(* IEC 61131-3 sources: 2026_Projet_YGO_ExcavatriceDragage/TOOLS/TEST_AUTO_CI/WORKING_COPY/tests (part 2) *)

(* ---- test_fb_cycle_negative.st ---- *)
SETUP
VAR
    FB : FB_Cycle;
    SampleCount : INT := 0;
END_VAR
END_SETUP

(* =====================================================================
   Harnais de TESTS NÉGATIFS — exécuté sur CODE/G_CYCLE/FB_Cycle.st (ORIGINAL).
   Chaque test DOIT ÉCHOUER sur l'original pour prouver la présence du défaut.
   Exclus de la suite verte (tests négatifs, exigence T3/T4 plan T171).
   ===================================================================== *)

TEST 'NEG-F1 : X11 ouverture benne commandee (doit ECHOUER sur original)'
    (* Atteindre X11 puis vérifier que BucketCmd.Open est TRUE quand le manche est défléchi.
       Sur l'original (read-before-write), Open reste FALSE -> ce test échoue. *)
    (* X0 -> X1 *)
    FB(Enable := TRUE, Reset := FALSE, PowerContactorEngaged := TRUE, Mode := E_Mode.SEMI_AUTO,
       DeadmanArmed := TRUE, CycleMotionPermit := TRUE, HeartbeatIhmOk := TRUE,
       StartCycle := TRUE, SelTarget := 3, SetDepthM := -10.0, SetOffsetM := 0.0,
       LimitLegalDepthM := -10.5, CableLimitM1AscentM := 7.0,
       SpeedMismatchThresholdMps := 0.0, SpeedMismatchTimeout := T#0ms,
       HomedM1 := TRUE, HomedM2 := TRUE, TopPositionSensor := TRUE, HomingRequest := FALSE,
       M1_CablePosM := 7.0, M2_CablePosM := 7.0, M1_MeasuredSpeedMps := 0.0, M2_MeasuredSpeedMps := 0.0,
       KoboldContactFond := FALSE, WinchSyncError := FALSE, WinchSyncDeltaM := 0.0,
       Translation_At_P1 := FALSE, Translation_At_Tremie := FALSE, Translation_At_Maintenance := FALSE,
       Translation_Busy := FALSE, Translation_Done := FALSE,
       Benne_Busy := FALSE, Benne_Done := FALSE, Benne_IsOpen := FALSE, Benne_IsClosed := TRUE, Benne_IsRoughlyClosed := TRUE,
       SampleCount := SampleCount);
    (* X1 -> X2 *)
    FB(Enable := TRUE, Reset := FALSE, PowerContactorEngaged := TRUE, Mode := E_Mode.SEMI_AUTO,
       DeadmanArmed := TRUE, CycleMotionPermit := TRUE, HeartbeatIhmOk := TRUE,
       StartCycle := FALSE, SelTarget := 3, SetDepthM := -10.0, SetOffsetM := 0.0,
       LimitLegalDepthM := -10.5, CableLimitM1AscentM := 7.0,
       SpeedMismatchThresholdMps := 0.0, SpeedMismatchTimeout := T#0ms,
       HomedM1 := TRUE, HomedM2 := TRUE, TopPositionSensor := TRUE, HomingRequest := FALSE,
       M1_CablePosM := 7.0, M2_CablePosM := 7.0, M1_MeasuredSpeedMps := 0.0, M2_MeasuredSpeedMps := 0.0,
       KoboldContactFond := FALSE, WinchSyncError := FALSE, WinchSyncDeltaM := 0.0,
       Translation_At_P1 := FALSE, Translation_At_Tremie := FALSE, Translation_At_Maintenance := FALSE,
       Translation_Busy := FALSE, Translation_Done := FALSE,
       Benne_Busy := FALSE, Benne_Done := FALSE, Benne_IsOpen := FALSE, Benne_IsClosed := TRUE, Benne_IsRoughlyClosed := TRUE,
       SampleCount := SampleCount);
    (* X2 -> X3 *)
    FB(Enable := TRUE, Reset := FALSE, PowerContactorEngaged := TRUE, Mode := E_Mode.SEMI_AUTO,
       DeadmanArmed := TRUE, CycleMotionPermit := TRUE, HeartbeatIhmOk := TRUE,
       StartCycle := FALSE, SelTarget := 3, SetDepthM := -10.0, SetOffsetM := 0.0,
       LimitLegalDepthM := -10.5, CableLimitM1AscentM := 7.0,
       SpeedMismatchThresholdMps := 0.0, SpeedMismatchTimeout := T#0ms,
       HomedM1 := TRUE, HomedM2 := TRUE, TopPositionSensor := TRUE, HomingRequest := FALSE,
       M1_CablePosM := 7.0, M2_CablePosM := 7.0, M1_MeasuredSpeedMps := 0.0, M2_MeasuredSpeedMps := 0.0,
       KoboldContactFond := FALSE, WinchSyncError := FALSE, WinchSyncDeltaM := 0.0,
       Translation_At_P1 := TRUE, Translation_At_Tremie := FALSE, Translation_At_Maintenance := FALSE,
       Translation_Busy := FALSE, Translation_Done := TRUE,
       Benne_Busy := FALSE, Benne_Done := FALSE, Benne_IsOpen := FALSE, Benne_IsClosed := TRUE, Benne_IsRoughlyClosed := TRUE,
       SampleCount := SampleCount);
    (* X3 -> X4 *)
    FB(Enable := TRUE, Reset := FALSE, PowerContactorEngaged := TRUE, Mode := E_Mode.SEMI_AUTO,
       DeadmanArmed := TRUE, CycleMotionPermit := TRUE, HeartbeatIhmOk := TRUE,
       StartCycle := FALSE, SelTarget := 3, SetDepthM := -10.0, SetOffsetM := 0.0,
       LimitLegalDepthM := -10.5, CableLimitM1AscentM := 7.0,
       SpeedMismatchThresholdMps := 0.0, SpeedMismatchTimeout := T#0ms,
       HomedM1 := TRUE, HomedM2 := TRUE, TopPositionSensor := TRUE, HomingRequest := FALSE,
       M1_CablePosM := 7.0, M2_CablePosM := 7.0, M1_MeasuredSpeedMps := 0.0, M2_MeasuredSpeedMps := 0.0,
       KoboldContactFond := FALSE, WinchSyncError := FALSE, WinchSyncDeltaM := 0.0,
       Translation_At_P1 := TRUE, Translation_At_Tremie := FALSE, Translation_At_Maintenance := FALSE,
       Translation_Busy := FALSE, Translation_Done := TRUE,
       Benne_Busy := FALSE, Benne_Done := FALSE, Benne_IsOpen := TRUE, Benne_IsClosed := FALSE, Benne_IsRoughlyClosed := FALSE,
       SampleCount := SampleCount);
    (* X4 -> X5 *)
    FB(Enable := TRUE, Reset := FALSE, PowerContactorEngaged := TRUE, Mode := E_Mode.SEMI_AUTO,
       DeadmanArmed := TRUE, CycleMotionPermit := TRUE, HeartbeatIhmOk := TRUE,
       StartCycle := FALSE, SelTarget := 3, SetDepthM := -10.0, SetOffsetM := 0.0,
       LimitLegalDepthM := -10.5, CableLimitM1AscentM := 7.0,
       SpeedMismatchThresholdMps := 0.0, SpeedMismatchTimeout := T#0ms,
       HomedM1 := TRUE, HomedM2 := TRUE, TopPositionSensor := TRUE, HomingRequest := FALSE,
       M1_CablePosM := -10.0, M2_CablePosM := -10.0, M1_MeasuredSpeedMps := 0.0, M2_MeasuredSpeedMps := 0.0,
       KoboldContactFond := TRUE, WinchSyncError := FALSE, WinchSyncDeltaM := 0.0,
       Translation_At_P1 := TRUE, Translation_At_Tremie := FALSE, Translation_At_Maintenance := FALSE,
       Translation_Busy := FALSE, Translation_Done := TRUE,
       Benne_Busy := FALSE, Benne_Done := FALSE, Benne_IsOpen := TRUE, Benne_IsClosed := FALSE, Benne_IsRoughlyClosed := FALSE,
       SampleCount := SampleCount);
    (* X5 -> X6 *)
    FB(Enable := TRUE, Reset := FALSE, PowerContactorEngaged := TRUE, Mode := E_Mode.SEMI_AUTO,
       DeadmanArmed := TRUE, CycleMotionPermit := TRUE, HeartbeatIhmOk := TRUE,
       StartCycle := FALSE, SelTarget := 3, SetDepthM := -10.0, SetOffsetM := 0.0,
       LimitLegalDepthM := -10.5, CableLimitM1AscentM := 7.0,
       SpeedMismatchThresholdMps := 0.0, SpeedMismatchTimeout := T#0ms,
       HomedM1 := TRUE, HomedM2 := TRUE, TopPositionSensor := TRUE, HomingRequest := FALSE,
       M1_CablePosM := -9.5, M2_CablePosM := -9.5, M1_MeasuredSpeedMps := 0.0, M2_MeasuredSpeedMps := 0.0,
       KoboldContactFond := FALSE, WinchSyncError := FALSE, WinchSyncDeltaM := 0.0,
       Translation_At_P1 := TRUE, Translation_At_Tremie := FALSE, Translation_At_Maintenance := FALSE,
       Translation_Busy := FALSE, Translation_Done := TRUE,
       Benne_Busy := FALSE, Benne_Done := FALSE, Benne_IsOpen := TRUE, Benne_IsClosed := FALSE, Benne_IsRoughlyClosed := FALSE,
       SampleCount := SampleCount);
    (* X6 -> X7 *)
    FB(Enable := TRUE, Reset := FALSE, PowerContactorEngaged := TRUE, Mode := E_Mode.SEMI_AUTO,
       DeadmanArmed := TRUE, CycleMotionPermit := TRUE, HeartbeatIhmOk := TRUE,
       StartCycle := FALSE, SelTarget := 3, SetDepthM := -10.0, SetOffsetM := 0.0,
       LimitLegalDepthM := -10.5, CableLimitM1AscentM := 7.0,
       SpeedMismatchThresholdMps := 0.0, SpeedMismatchTimeout := T#0ms,
       HomedM1 := TRUE, HomedM2 := TRUE, TopPositionSensor := TRUE, HomingRequest := FALSE,
       M1_CablePosM := -9.5, M2_CablePosM := -9.5, M1_MeasuredSpeedMps := 0.0, M2_MeasuredSpeedMps := 0.0,
       KoboldContactFond := FALSE, WinchSyncError := FALSE, WinchSyncDeltaM := 0.0,
       Translation_At_P1 := TRUE, Translation_At_Tremie := FALSE, Translation_At_Maintenance := FALSE,
       Translation_Busy := FALSE, Translation_Done := TRUE,
       Benne_Busy := FALSE, Benne_Done := TRUE, Benne_IsOpen := FALSE, Benne_IsClosed := TRUE, Benne_IsRoughlyClosed := TRUE,
       SampleCount := SampleCount);
    (* X7 -> X8 *)
    FB(Enable := TRUE, Reset := FALSE, PowerContactorEngaged := TRUE, Mode := E_Mode.SEMI_AUTO,
       DeadmanArmed := TRUE, CycleMotionPermit := TRUE, HeartbeatIhmOk := TRUE,
       StartCycle := FALSE, SelTarget := 3, SetDepthM := -10.0, SetOffsetM := 0.0,
       LimitLegalDepthM := -10.5, CableLimitM1AscentM := 7.0,
       SpeedMismatchThresholdMps := 0.0, SpeedMismatchTimeout := T#0ms,
       HomedM1 := TRUE, HomedM2 := TRUE, TopPositionSensor := TRUE, HomingRequest := FALSE,
       M1_CablePosM := -8.0, M2_CablePosM := -8.0, M1_MeasuredSpeedMps := 0.0, M2_MeasuredSpeedMps := 0.0,
       KoboldContactFond := FALSE, WinchSyncError := FALSE, WinchSyncDeltaM := 0.0,
       Translation_At_P1 := TRUE, Translation_At_Tremie := FALSE, Translation_At_Maintenance := FALSE,
       Translation_Busy := FALSE, Translation_Done := TRUE,
       Benne_Busy := FALSE, Benne_Done := TRUE, Benne_IsOpen := FALSE, Benne_IsClosed := TRUE, Benne_IsRoughlyClosed := TRUE,
       SampleCount := SampleCount);
    (* X8 -> X9 *)
    FB(Enable := TRUE, Reset := FALSE, PowerContactorEngaged := TRUE, Mode := E_Mode.SEMI_AUTO,
       DeadmanArmed := TRUE, CycleMotionPermit := TRUE, HeartbeatIhmOk := TRUE,
       StartCycle := FALSE, SelTarget := 3, SetDepthM := -10.0, SetOffsetM := 0.0,
       LimitLegalDepthM := -10.5, CableLimitM1AscentM := 7.0,
       SpeedMismatchThresholdMps := 0.0, SpeedMismatchTimeout := T#0ms,
       HomedM1 := TRUE, HomedM2 := TRUE, TopPositionSensor := TRUE, HomingRequest := FALSE,
       M1_CablePosM := 7.0, M2_CablePosM := 7.0, M1_MeasuredSpeedMps := 0.0, M2_MeasuredSpeedMps := 0.0,
       KoboldContactFond := FALSE, WinchSyncError := FALSE, WinchSyncDeltaM := 0.0,
       Translation_At_P1 := TRUE, Translation_At_Tremie := FALSE, Translation_At_Maintenance := FALSE,
       Translation_Busy := FALSE, Translation_Done := TRUE,
       Benne_Busy := FALSE, Benne_Done := TRUE, Benne_IsOpen := FALSE, Benne_IsClosed := TRUE, Benne_IsRoughlyClosed := TRUE,
       SampleCount := SampleCount);
    (* X9 (démarre timer) *)
    FB(Enable := TRUE, Reset := FALSE, PowerContactorEngaged := TRUE, Mode := E_Mode.SEMI_AUTO,
       DeadmanArmed := TRUE, CycleMotionPermit := TRUE, HeartbeatIhmOk := TRUE,
       StartCycle := FALSE, SelTarget := 3, SetDepthM := -10.0, SetOffsetM := 0.0,
       LimitLegalDepthM := -10.5, CableLimitM1AscentM := 7.0,
       SpeedMismatchThresholdMps := 0.0, SpeedMismatchTimeout := T#0ms,
       HomedM1 := TRUE, HomedM2 := TRUE, TopPositionSensor := TRUE, HomingRequest := FALSE,
       M1_CablePosM := 7.0, M2_CablePosM := 7.0, M1_MeasuredSpeedMps := 0.0, M2_MeasuredSpeedMps := 0.0,
       KoboldContactFond := FALSE, WinchSyncError := FALSE, WinchSyncDeltaM := 0.0,
       Translation_At_P1 := TRUE, Translation_At_Tremie := FALSE, Translation_At_Maintenance := FALSE,
       Translation_Busy := FALSE, Translation_Done := TRUE,
       Benne_Busy := FALSE, Benne_Done := TRUE, Benne_IsOpen := FALSE, Benne_IsClosed := TRUE, Benne_IsRoughlyClosed := TRUE,
       SampleCount := SampleCount);
    (* X9 -> X10 *)
    ADVANCE_TIME(5000000000);
    FB(Enable := TRUE, Reset := FALSE, PowerContactorEngaged := TRUE, Mode := E_Mode.SEMI_AUTO,
       DeadmanArmed := TRUE, CycleMotionPermit := TRUE, HeartbeatIhmOk := TRUE,
       StartCycle := FALSE, SelTarget := 3, SetDepthM := -10.0, SetOffsetM := 0.0,
       LimitLegalDepthM := -10.5, CableLimitM1AscentM := 7.0,
       SpeedMismatchThresholdMps := 0.0, SpeedMismatchTimeout := T#0ms,
       HomedM1 := TRUE, HomedM2 := TRUE, TopPositionSensor := TRUE, HomingRequest := FALSE,
       M1_CablePosM := 7.0, M2_CablePosM := 7.0, M1_MeasuredSpeedMps := 0.0, M2_MeasuredSpeedMps := 0.0,
       KoboldContactFond := FALSE, WinchSyncError := FALSE, WinchSyncDeltaM := 0.0,
       Translation_At_P1 := TRUE, Translation_At_Tremie := FALSE, Translation_At_Maintenance := FALSE,
       Translation_Busy := FALSE, Translation_Done := TRUE,
       Benne_Busy := FALSE, Benne_Done := TRUE, Benne_IsOpen := FALSE, Benne_IsClosed := TRUE, Benne_IsRoughlyClosed := TRUE,
       SampleCount := SampleCount);
    (* X10 -> X11 *)
    FB(Enable := TRUE, Reset := FALSE, PowerContactorEngaged := TRUE, Mode := E_Mode.SEMI_AUTO,
       DeadmanArmed := TRUE, CycleMotionPermit := TRUE, HeartbeatIhmOk := TRUE,
       StartCycle := FALSE, SelTarget := 3, SetDepthM := -10.0, SetOffsetM := 0.0,
       LimitLegalDepthM := -10.5, CableLimitM1AscentM := 7.0,
       SpeedMismatchThresholdMps := 0.0, SpeedMismatchTimeout := T#0ms,
       HomedM1 := TRUE, HomedM2 := TRUE, TopPositionSensor := TRUE, HomingRequest := FALSE,
       M1_CablePosM := 7.0, M2_CablePosM := 7.0, M1_MeasuredSpeedMps := 0.0, M2_MeasuredSpeedMps := 0.0,
       KoboldContactFond := FALSE, WinchSyncError := FALSE, WinchSyncDeltaM := 0.0,
       Translation_At_P1 := FALSE, Translation_At_Tremie := TRUE, Translation_At_Maintenance := FALSE,
       Translation_Busy := FALSE, Translation_Done := TRUE,
       Benne_Busy := FALSE, Benne_Done := TRUE, Benne_IsOpen := FALSE, Benne_IsClosed := TRUE, Benne_IsRoughlyClosed := TRUE,
       SampleCount := SampleCount);
    (* X11 : manche défléchi, benne PAS encore ouverte -> BucketCmd.Open doit être TRUE
       (sur original : FALSE, read-before-write). Benne_Done=FALSE/IsOpen=FALSE pour ne PAS
       déclencher la transition X11->X13 dans ce scan. *)
    FB(Enable := TRUE, Reset := FALSE, PowerContactorEngaged := TRUE, Mode := E_Mode.SEMI_AUTO,
       DeadmanArmed := TRUE, CycleMotionPermit := TRUE, HeartbeatIhmOk := TRUE,
       StartCycle := FALSE, SelTarget := 3, SetDepthM := -10.0, SetOffsetM := 0.0,
       LimitLegalDepthM := -10.5, CableLimitM1AscentM := 7.0,
       SpeedMismatchThresholdMps := 0.0, SpeedMismatchTimeout := T#0ms,
       HomedM1 := TRUE, HomedM2 := TRUE, TopPositionSensor := TRUE, HomingRequest := FALSE,
       M1_CablePosM := 7.0, M2_CablePosM := 7.0, M1_MeasuredSpeedMps := 0.0, M2_MeasuredSpeedMps := 0.0,
       KoboldContactFond := FALSE, WinchSyncError := FALSE, WinchSyncDeltaM := 0.0,
       Translation_At_P1 := FALSE, Translation_At_Tremie := TRUE, Translation_At_Maintenance := FALSE,
       Translation_Busy := FALSE, Translation_Done := TRUE,
       Benne_Busy := FALSE, Benne_Done := FALSE, Benne_IsOpen := FALSE, Benne_IsClosed := TRUE, Benne_IsRoughlyClosed := TRUE,
       SampleCount := SampleCount);
    ASSERT_TRUE(FB.BucketCmd.Open, 'NEG-F1: ouverture benne commandée en X11 (échoue sur original)');
END_TEST

TEST 'NEG-F2 : SampleCount +1 strict sur X13 multi-scan (doit ECHOUER sur original)'
    (* Atteindre X13 puis rester 2 scans. Sur l'original, SampleCount augmente à chaque scan
       (2 au lieu de 1) -> ce test échoue. *)
    (* X0 -> X1 *)
    FB(Enable := TRUE, Reset := FALSE, PowerContactorEngaged := TRUE, Mode := E_Mode.SEMI_AUTO,
       DeadmanArmed := TRUE, CycleMotionPermit := TRUE, HeartbeatIhmOk := TRUE,
       StartCycle := TRUE, SelTarget := 3, SetDepthM := -10.0, SetOffsetM := 0.0,
       LimitLegalDepthM := -10.5, CableLimitM1AscentM := 7.0,
       SpeedMismatchThresholdMps := 0.0, SpeedMismatchTimeout := T#0ms,
       HomedM1 := TRUE, HomedM2 := TRUE, TopPositionSensor := TRUE, HomingRequest := FALSE,
       M1_CablePosM := 7.0, M2_CablePosM := 7.0, M1_MeasuredSpeedMps := 0.0, M2_MeasuredSpeedMps := 0.0,
       KoboldContactFond := FALSE, WinchSyncError := FALSE, WinchSyncDeltaM := 0.0,
       Translation_At_P1 := FALSE, Translation_At_Tremie := FALSE, Translation_At_Maintenance := FALSE,
       Translation_Busy := FALSE, Translation_Done := FALSE,
       Benne_Busy := FALSE, Benne_Done := FALSE, Benne_IsOpen := FALSE, Benne_IsClosed := TRUE, Benne_IsRoughlyClosed := TRUE,
       SampleCount := SampleCount);
    (* X1 -> X2 *)
    FB(Enable := TRUE, Reset := FALSE, PowerContactorEngaged := TRUE, Mode := E_Mode.SEMI_AUTO,
       DeadmanArmed := TRUE, CycleMotionPermit := TRUE, HeartbeatIhmOk := TRUE,
       StartCycle := FALSE, SelTarget := 3, SetDepthM := -10.0, SetOffsetM := 0.0,
       LimitLegalDepthM := -10.5, CableLimitM1AscentM := 7.0,
       SpeedMismatchThresholdMps := 0.0, SpeedMismatchTimeout := T#0ms,
       HomedM1 := TRUE, HomedM2 := TRUE, TopPositionSensor := TRUE, HomingRequest := FALSE,
       M1_CablePosM := 7.0, M2_CablePosM := 7.0, M1_MeasuredSpeedMps := 0.0, M2_MeasuredSpeedMps := 0.0,
       KoboldContactFond := FALSE, WinchSyncError := FALSE, WinchSyncDeltaM := 0.0,
       Translation_At_P1 := FALSE, Translation_At_Tremie := FALSE, Translation_At_Maintenance := FALSE,
       Translation_Busy := FALSE, Translation_Done := FALSE,
       Benne_Busy := FALSE, Benne_Done := FALSE, Benne_IsOpen := FALSE, Benne_IsClosed := TRUE, Benne_IsRoughlyClosed := TRUE,
       SampleCount := SampleCount);
    (* X2 -> X3 *)
    FB(Enable := TRUE, Reset := FALSE, PowerContactorEngaged := TRUE, Mode := E_Mode.SEMI_AUTO,
       DeadmanArmed := TRUE, CycleMotionPermit := TRUE, HeartbeatIhmOk := TRUE,
       StartCycle := FALSE, SelTarget := 3, SetDepthM := -10.0, SetOffsetM := 0.0,
       LimitLegalDepthM := -10.5, CableLimitM1AscentM := 7.0,
       SpeedMismatchThresholdMps := 0.0, SpeedMismatchTimeout := T#0ms,
       HomedM1 := TRUE, HomedM2 := TRUE, TopPositionSensor := TRUE, HomingRequest := FALSE,
       M1_CablePosM := 7.0, M2_CablePosM := 7.0, M1_MeasuredSpeedMps := 0.0, M2_MeasuredSpeedMps := 0.0,
       KoboldContactFond := FALSE, WinchSyncError := FALSE, WinchSyncDeltaM := 0.0,
       Translation_At_P1 := TRUE, Translation_At_Tremie := FALSE, Translation_At_Maintenance := FALSE,
       Translation_Busy := FALSE, Translation_Done := TRUE,
       Benne_Busy := FALSE, Benne_Done := FALSE, Benne_IsOpen := FALSE, Benne_IsClosed := TRUE, Benne_IsRoughlyClosed := TRUE,
       SampleCount := SampleCount);
    (* X3 -> X4 *)
    FB(Enable := TRUE, Reset := FALSE, PowerContactorEngaged := TRUE, Mode := E_Mode.SEMI_AUTO,
       DeadmanArmed := TRUE, CycleMotionPermit := TRUE, HeartbeatIhmOk := TRUE,
       StartCycle := FALSE, SelTarget := 3, SetDepthM := -10.0, SetOffsetM := 0.0,
       LimitLegalDepthM := -10.5, CableLimitM1AscentM := 7.0,
       SpeedMismatchThresholdMps := 0.0, SpeedMismatchTimeout := T#0ms,
       HomedM1 := TRUE, HomedM2 := TRUE, TopPositionSensor := TRUE, HomingRequest := FALSE,
       M1_CablePosM := 7.0, M2_CablePosM := 7.0, M1_MeasuredSpeedMps := 0.0, M2_MeasuredSpeedMps := 0.0,
       KoboldContactFond := FALSE, WinchSyncError := FALSE, WinchSyncDeltaM := 0.0,
       Translation_At_P1 := TRUE, Translation_At_Tremie := FALSE, Translation_At_Maintenance := FALSE,
       Translation_Busy := FALSE, Translation_Done := TRUE,
       Benne_Busy := FALSE, Benne_Done := FALSE, Benne_IsOpen := TRUE, Benne_IsClosed := FALSE, Benne_IsRoughlyClosed := FALSE,
       SampleCount := SampleCount);
    (* X4 -> X5 *)
    FB(Enable := TRUE, Reset := FALSE, PowerContactorEngaged := TRUE, Mode := E_Mode.SEMI_AUTO,
       DeadmanArmed := TRUE, CycleMotionPermit := TRUE, HeartbeatIhmOk := TRUE,
       StartCycle := FALSE, SelTarget := 3, SetDepthM := -10.0, SetOffsetM := 0.0,
       LimitLegalDepthM := -10.5, CableLimitM1AscentM := 7.0,
       SpeedMismatchThresholdMps := 0.0, SpeedMismatchTimeout := T#0ms,
       HomedM1 := TRUE, HomedM2 := TRUE, TopPositionSensor := TRUE, HomingRequest := FALSE,
       M1_CablePosM := -10.0, M2_CablePosM := -10.0, M1_MeasuredSpeedMps := 0.0, M2_MeasuredSpeedMps := 0.0,
       KoboldContactFond := TRUE, WinchSyncError := FALSE, WinchSyncDeltaM := 0.0,
       Translation_At_P1 := TRUE, Translation_At_Tremie := FALSE, Translation_At_Maintenance := FALSE,
       Translation_Busy := FALSE, Translation_Done := TRUE,
       Benne_Busy := FALSE, Benne_Done := FALSE, Benne_IsOpen := TRUE, Benne_IsClosed := FALSE, Benne_IsRoughlyClosed := FALSE,
       SampleCount := SampleCount);
    (* X5 -> X6 *)
    FB(Enable := TRUE, Reset := FALSE, PowerContactorEngaged := TRUE, Mode := E_Mode.SEMI_AUTO,
       DeadmanArmed := TRUE, CycleMotionPermit := TRUE, HeartbeatIhmOk := TRUE,
       StartCycle := FALSE, SelTarget := 3, SetDepthM := -10.0, SetOffsetM := 0.0,
       LimitLegalDepthM := -10.5, CableLimitM1AscentM := 7.0,
       SpeedMismatchThresholdMps := 0.0, SpeedMismatchTimeout := T#0ms,
       HomedM1 := TRUE, HomedM2 := TRUE, TopPositionSensor := TRUE, HomingRequest := FALSE,
       M1_CablePosM := -9.5, M2_CablePosM := -9.5, M1_MeasuredSpeedMps := 0.0, M2_MeasuredSpeedMps := 0.0,
       KoboldContactFond := FALSE, WinchSyncError := FALSE, WinchSyncDeltaM := 0.0,
       Translation_At_P1 := TRUE, Translation_At_Tremie := FALSE, Translation_At_Maintenance := FALSE,
       Translation_Busy := FALSE, Translation_Done := TRUE,
       Benne_Busy := FALSE, Benne_Done := FALSE, Benne_IsOpen := TRUE, Benne_IsClosed := FALSE, Benne_IsRoughlyClosed := FALSE,
       SampleCount := SampleCount);
    (* X6 -> X7 *)
    FB(Enable := TRUE, Reset := FALSE, PowerContactorEngaged := TRUE, Mode := E_Mode.SEMI_AUTO,
       DeadmanArmed := TRUE, CycleMotionPermit := TRUE, HeartbeatIhmOk := TRUE,
       StartCycle := FALSE, SelTarget := 3, SetDepthM := -10.0, SetOffsetM := 0.0,
       LimitLegalDepthM := -10.5, CableLimitM1AscentM := 7.0,
       SpeedMismatchThresholdMps := 0.0, SpeedMismatchTimeout := T#0ms,
       HomedM1 := TRUE, HomedM2 := TRUE, TopPositionSensor := TRUE, HomingRequest := FALSE,
       M1_CablePosM := -9.5, M2_CablePosM := -9.5, M1_MeasuredSpeedMps := 0.0, M2_MeasuredSpeedMps := 0.0,
       KoboldContactFond := FALSE, WinchSyncError := FALSE, WinchSyncDeltaM := 0.0,
       Translation_At_P1 := TRUE, Translation_At_Tremie := FALSE, Translation_At_Maintenance := FALSE,
       Translation_Busy := FALSE, Translation_Done := TRUE,
       Benne_Busy := FALSE, Benne_Done := TRUE, Benne_IsOpen := FALSE, Benne_IsClosed := TRUE, Benne_IsRoughlyClosed := TRUE,
       SampleCount := SampleCount);
    (* X7 -> X8 *)
    FB(Enable := TRUE, Reset := FALSE, PowerContactorEngaged := TRUE, Mode := E_Mode.SEMI_AUTO,
       DeadmanArmed := TRUE, CycleMotionPermit := TRUE, HeartbeatIhmOk := TRUE,
       StartCycle := FALSE, SelTarget := 3, SetDepthM := -10.0, SetOffsetM := 0.0,
       LimitLegalDepthM := -10.5, CableLimitM1AscentM := 7.0,
       SpeedMismatchThresholdMps := 0.0, SpeedMismatchTimeout := T#0ms,
       HomedM1 := TRUE, HomedM2 := TRUE, TopPositionSensor := TRUE, HomingRequest := FALSE,
       M1_CablePosM := -8.0, M2_CablePosM := -8.0, M1_MeasuredSpeedMps := 0.0, M2_MeasuredSpeedMps := 0.0,
       KoboldContactFond := FALSE, WinchSyncError := FALSE, WinchSyncDeltaM := 0.0,
       Translation_At_P1 := TRUE, Translation_At_Tremie := FALSE, Translation_At_Maintenance := FALSE,
       Translation_Busy := FALSE, Translation_Done := TRUE,
       Benne_Busy := FALSE, Benne_Done := TRUE, Benne_IsOpen := FALSE, Benne_IsClosed := TRUE, Benne_IsRoughlyClosed := TRUE,
       SampleCount := SampleCount);
    (* X8 -> X9 *)
    FB(Enable := TRUE, Reset := FALSE, PowerContactorEngaged := TRUE, Mode := E_Mode.SEMI_AUTO,
       DeadmanArmed := TRUE, CycleMotionPermit := TRUE, HeartbeatIhmOk := TRUE,
       StartCycle := FALSE, SelTarget := 3, SetDepthM := -10.0, SetOffsetM := 0.0,
       LimitLegalDepthM := -10.5, CableLimitM1AscentM := 7.0,
       SpeedMismatchThresholdMps := 0.0, SpeedMismatchTimeout := T#0ms,
       HomedM1 := TRUE, HomedM2 := TRUE, TopPositionSensor := TRUE, HomingRequest := FALSE,
       M1_CablePosM := 7.0, M2_CablePosM := 7.0, M1_MeasuredSpeedMps := 0.0, M2_MeasuredSpeedMps := 0.0,
       KoboldContactFond := FALSE, WinchSyncError := FALSE, WinchSyncDeltaM := 0.0,
       Translation_At_P1 := TRUE, Translation_At_Tremie := FALSE, Translation_At_Maintenance := FALSE,
       Translation_Busy := FALSE, Translation_Done := TRUE,
       Benne_Busy := FALSE, Benne_Done := TRUE, Benne_IsOpen := FALSE, Benne_IsClosed := TRUE, Benne_IsRoughlyClosed := TRUE,
       SampleCount := SampleCount);
    (* X9 (démarre timer) *)
    FB(Enable := TRUE, Reset := FALSE, PowerContactorEngaged := TRUE, Mode := E_Mode.SEMI_AUTO,
       DeadmanArmed := TRUE, CycleMotionPermit := TRUE, HeartbeatIhmOk := TRUE,
       StartCycle := FALSE, SelTarget := 3, SetDepthM := -10.0, SetOffsetM := 0.0,
       LimitLegalDepthM := -10.5, CableLimitM1AscentM := 7.0,
       SpeedMismatchThresholdMps := 0.0, SpeedMismatchTimeout := T#0ms,
       HomedM1 := TRUE, HomedM2 := TRUE, TopPositionSensor := TRUE, HomingRequest := FALSE,
       M1_CablePosM := 7.0, M2_CablePosM := 7.0, M1_MeasuredSpeedMps := 0.0, M2_MeasuredSpeedMps := 0.0,
       KoboldContactFond := FALSE, WinchSyncError := FALSE, WinchSyncDeltaM := 0.0,
       Translation_At_P1 := TRUE, Translation_At_Tremie := FALSE, Translation_At_Maintenance := FALSE,
       Translation_Busy := FALSE, Translation_Done := TRUE,
       Benne_Busy := FALSE, Benne_Done := TRUE, Benne_IsOpen := FALSE, Benne_IsClosed := TRUE, Benne_IsRoughlyClosed := TRUE,
       SampleCount := SampleCount);
    (* X9 -> X10 *)
    ADVANCE_TIME(5000000000);
    FB(Enable := TRUE, Reset := FALSE, PowerContactorEngaged := TRUE, Mode := E_Mode.SEMI_AUTO,
       DeadmanArmed := TRUE, CycleMotionPermit := TRUE, HeartbeatIhmOk := TRUE,
       StartCycle := FALSE, SelTarget := 3, SetDepthM := -10.0, SetOffsetM := 0.0,
       LimitLegalDepthM := -10.5, CableLimitM1AscentM := 7.0,
       SpeedMismatchThresholdMps := 0.0, SpeedMismatchTimeout := T#0ms,
       HomedM1 := TRUE, HomedM2 := TRUE, TopPositionSensor := TRUE, HomingRequest := FALSE,
       M1_CablePosM := 7.0, M2_CablePosM := 7.0, M1_MeasuredSpeedMps := 0.0, M2_MeasuredSpeedMps := 0.0,
       KoboldContactFond := FALSE, WinchSyncError := FALSE, WinchSyncDeltaM := 0.0,
       Translation_At_P1 := TRUE, Translation_At_Tremie := FALSE, Translation_At_Maintenance := FALSE,
       Translation_Busy := FALSE, Translation_Done := TRUE,
       Benne_Busy := FALSE, Benne_Done := TRUE, Benne_IsOpen := FALSE, Benne_IsClosed := TRUE, Benne_IsRoughlyClosed := TRUE,
       SampleCount := SampleCount);
    (* X10 -> X11 *)
    FB(Enable := TRUE, Reset := FALSE, PowerContactorEngaged := TRUE, Mode := E_Mode.SEMI_AUTO,
       DeadmanArmed := TRUE, CycleMotionPermit := TRUE, HeartbeatIhmOk := TRUE,
       StartCycle := FALSE, SelTarget := 3, SetDepthM := -10.0, SetOffsetM := 0.0,
       LimitLegalDepthM := -10.5, CableLimitM1AscentM := 7.0,
       SpeedMismatchThresholdMps := 0.0, SpeedMismatchTimeout := T#0ms,
       HomedM1 := TRUE, HomedM2 := TRUE, TopPositionSensor := TRUE, HomingRequest := FALSE,
       M1_CablePosM := 7.0, M2_CablePosM := 7.0, M1_MeasuredSpeedMps := 0.0, M2_MeasuredSpeedMps := 0.0,
       KoboldContactFond := FALSE, WinchSyncError := FALSE, WinchSyncDeltaM := 0.0,
       Translation_At_P1 := FALSE, Translation_At_Tremie := TRUE, Translation_At_Maintenance := FALSE,
       Translation_Busy := FALSE, Translation_Done := TRUE,
       Benne_Busy := FALSE, Benne_Done := TRUE, Benne_IsOpen := FALSE, Benne_IsClosed := TRUE, Benne_IsRoughlyClosed := TRUE,
       SampleCount := SampleCount);
    (* X11 -> X13 *)
    FB(Enable := TRUE, Reset := FALSE, PowerContactorEngaged := TRUE, Mode := E_Mode.SEMI_AUTO,
       DeadmanArmed := TRUE, CycleMotionPermit := TRUE, HeartbeatIhmOk := TRUE,
       StartCycle := FALSE, SelTarget := 3, SetDepthM := -10.0, SetOffsetM := 0.0,
       LimitLegalDepthM := -10.5, CableLimitM1AscentM := 7.0,
       SpeedMismatchThresholdMps := 0.0, SpeedMismatchTimeout := T#0ms,
       HomedM1 := TRUE, HomedM2 := TRUE, TopPositionSensor := TRUE, HomingRequest := FALSE,
       M1_CablePosM := 7.0, M2_CablePosM := 7.0, M1_MeasuredSpeedMps := 0.0, M2_MeasuredSpeedMps := 0.0,
       KoboldContactFond := FALSE, WinchSyncError := FALSE, WinchSyncDeltaM := 0.0,
       Translation_At_P1 := FALSE, Translation_At_Tremie := TRUE, Translation_At_Maintenance := FALSE,
       Translation_Busy := FALSE, Translation_Done := TRUE,
       Benne_Busy := FALSE, Benne_Done := TRUE, Benne_IsOpen := TRUE, Benne_IsClosed := FALSE, Benne_IsRoughlyClosed := FALSE,
       SampleCount := SampleCount);
    (* X13 (1er scan) *)
    FB(Enable := TRUE, Reset := FALSE, PowerContactorEngaged := TRUE, Mode := E_Mode.SEMI_AUTO,
       DeadmanArmed := TRUE, CycleMotionPermit := TRUE, HeartbeatIhmOk := TRUE,
       StartCycle := FALSE, SelTarget := 3, SetDepthM := -10.0, SetOffsetM := 0.0,
       LimitLegalDepthM := -10.5, CableLimitM1AscentM := 7.0,
       SpeedMismatchThresholdMps := 0.0, SpeedMismatchTimeout := T#0ms,
       HomedM1 := TRUE, HomedM2 := TRUE, TopPositionSensor := TRUE, HomingRequest := FALSE,
       M1_CablePosM := 7.0, M2_CablePosM := 7.0, M1_MeasuredSpeedMps := 0.0, M2_MeasuredSpeedMps := 0.0,
       KoboldContactFond := FALSE, WinchSyncError := FALSE, WinchSyncDeltaM := 0.0,
       Translation_At_P1 := FALSE, Translation_At_Tremie := TRUE, Translation_At_Maintenance := FALSE,
       Translation_Busy := FALSE, Translation_Done := TRUE,
       Benne_Busy := FALSE, Benne_Done := TRUE, Benne_IsOpen := TRUE, Benne_IsClosed := FALSE, Benne_IsRoughlyClosed := FALSE,
       SampleCount := SampleCount);
    (* X13 (2e scan) : SampleCount doit rester 1 (sur original : 2) *)
    FB(Enable := TRUE, Reset := FALSE, PowerContactorEngaged := TRUE, Mode := E_Mode.SEMI_AUTO,
       DeadmanArmed := TRUE, CycleMotionPermit := TRUE, HeartbeatIhmOk := TRUE,
       StartCycle := FALSE, SelTarget := 3, SetDepthM := -10.0, SetOffsetM := 0.0,
       LimitLegalDepthM := -10.5, CableLimitM1AscentM := 7.0,
       SpeedMismatchThresholdMps := 0.0, SpeedMismatchTimeout := T#0ms,
       HomedM1 := TRUE, HomedM2 := TRUE, TopPositionSensor := TRUE, HomingRequest := FALSE,
       M1_CablePosM := 7.0, M2_CablePosM := 7.0, M1_MeasuredSpeedMps := 0.0, M2_MeasuredSpeedMps := 0.0,
       KoboldContactFond := FALSE, WinchSyncError := FALSE, WinchSyncDeltaM := 0.0,
       Translation_At_P1 := FALSE, Translation_At_Tremie := TRUE, Translation_At_Maintenance := FALSE,
       Translation_Busy := FALSE, Translation_Done := TRUE,
       Benne_Busy := FALSE, Benne_Done := TRUE, Benne_IsOpen := TRUE, Benne_IsClosed := FALSE, Benne_IsRoughlyClosed := FALSE,
       SampleCount := SampleCount);
    (* X13 (3e scan) : SampleCount doit rester 1 (sur original : 3) — expose l'incrément abusif *)
    FB(Enable := TRUE, Reset := FALSE, PowerContactorEngaged := TRUE, Mode := E_Mode.SEMI_AUTO,
       DeadmanArmed := TRUE, CycleMotionPermit := TRUE, HeartbeatIhmOk := TRUE,
       StartCycle := FALSE, SelTarget := 3, SetDepthM := -10.0, SetOffsetM := 0.0,
       LimitLegalDepthM := -10.5, CableLimitM1AscentM := 7.0,
       SpeedMismatchThresholdMps := 0.0, SpeedMismatchTimeout := T#0ms,
       HomedM1 := TRUE, HomedM2 := TRUE, TopPositionSensor := TRUE, HomingRequest := FALSE,
       M1_CablePosM := 7.0, M2_CablePosM := 7.0, M1_MeasuredSpeedMps := 0.0, M2_MeasuredSpeedMps := 0.0,
       KoboldContactFond := FALSE, WinchSyncError := FALSE, WinchSyncDeltaM := 0.0,
       Translation_At_P1 := FALSE, Translation_At_Tremie := TRUE, Translation_At_Maintenance := FALSE,
       Translation_Busy := FALSE, Translation_Done := TRUE,
       Benne_Busy := FALSE, Benne_Done := TRUE, Benne_IsOpen := TRUE, Benne_IsClosed := FALSE, Benne_IsRoughlyClosed := FALSE,
       SampleCount := SampleCount);
    ASSERT_EQ(FB.SampleCount, 1, 'NEG-F2: SampleCount reste 1 au 3e scan en X13 (échoue sur original)');
END_TEST

TEST 'NEG-F6 : reprise consciente exigee apres bascule mode (doit ECHOUER sur original)'
    (* Atteindre X4, basculer MAINT, revenir SEMI_AUTO avec manche défléchi.
       Sur l'original, le mouvement reprend AUTOMATIQUEMENT (WinchM1Cmd.StartStop=TRUE).
       Sur la copie corrigée, il est neutralisé (F6). Ce test échoue sur l'original. *)
    (* X0 -> X1 *)
    FB(Enable := TRUE, Reset := FALSE, PowerContactorEngaged := TRUE, Mode := E_Mode.SEMI_AUTO,
       DeadmanArmed := TRUE, CycleMotionPermit := TRUE, HeartbeatIhmOk := TRUE,
       StartCycle := TRUE, SelTarget := 3, SetDepthM := -10.0, SetOffsetM := 0.0,
       LimitLegalDepthM := -10.5, CableLimitM1AscentM := 7.0,
       SpeedMismatchThresholdMps := 0.0, SpeedMismatchTimeout := T#0ms,
       HomedM1 := TRUE, HomedM2 := TRUE, TopPositionSensor := TRUE, HomingRequest := FALSE,
       M1_CablePosM := 7.0, M2_CablePosM := 7.0, M1_MeasuredSpeedMps := 0.0, M2_MeasuredSpeedMps := 0.0,
       KoboldContactFond := FALSE, WinchSyncError := FALSE, WinchSyncDeltaM := 0.0,
       Translation_At_P1 := FALSE, Translation_At_Tremie := FALSE, Translation_At_Maintenance := FALSE,
       Translation_Busy := FALSE, Translation_Done := FALSE,
       Benne_Busy := FALSE, Benne_Done := FALSE, Benne_IsOpen := FALSE, Benne_IsClosed := TRUE, Benne_IsRoughlyClosed := TRUE,
       SampleCount := SampleCount);
    (* X1 -> X2 *)
    FB(Enable := TRUE, Reset := FALSE, PowerContactorEngaged := TRUE, Mode := E_Mode.SEMI_AUTO,
       DeadmanArmed := TRUE, CycleMotionPermit := TRUE, HeartbeatIhmOk := TRUE,
       StartCycle := FALSE, SelTarget := 3, SetDepthM := -10.0, SetOffsetM := 0.0,
       LimitLegalDepthM := -10.5, CableLimitM1AscentM := 7.0,
       SpeedMismatchThresholdMps := 0.0, SpeedMismatchTimeout := T#0ms,
       HomedM1 := TRUE, HomedM2 := TRUE, TopPositionSensor := TRUE, HomingRequest := FALSE,
       M1_CablePosM := 7.0, M2_CablePosM := 7.0, M1_MeasuredSpeedMps := 0.0, M2_MeasuredSpeedMps := 0.0,
       KoboldContactFond := FALSE, WinchSyncError := FALSE, WinchSyncDeltaM := 0.0,
       Translation_At_P1 := FALSE, Translation_At_Tremie := FALSE, Translation_At_Maintenance := FALSE,
       Translation_Busy := FALSE, Translation_Done := FALSE,
       Benne_Busy := FALSE, Benne_Done := FALSE, Benne_IsOpen := FALSE, Benne_IsClosed := TRUE, Benne_IsRoughlyClosed := TRUE,
       SampleCount := SampleCount);
    (* X2 -> X3 *)
    FB(Enable := TRUE, Reset := FALSE, PowerContactorEngaged := TRUE, Mode := E_Mode.SEMI_AUTO,
       DeadmanArmed := TRUE, CycleMotionPermit := TRUE, HeartbeatIhmOk := TRUE,
       StartCycle := FALSE, SelTarget := 3, SetDepthM := -10.0, SetOffsetM := 0.0,
       LimitLegalDepthM := -10.5, CableLimitM1AscentM := 7.0,
       SpeedMismatchThresholdMps := 0.0, SpeedMismatchTimeout := T#0ms,
       HomedM1 := TRUE, HomedM2 := TRUE, TopPositionSensor := TRUE, HomingRequest := FALSE,
       M1_CablePosM := 7.0, M2_CablePosM := 7.0, M1_MeasuredSpeedMps := 0.0, M2_MeasuredSpeedMps := 0.0,
       KoboldContactFond := FALSE, WinchSyncError := FALSE, WinchSyncDeltaM := 0.0,
       Translation_At_P1 := TRUE, Translation_At_Tremie := FALSE, Translation_At_Maintenance := FALSE,
       Translation_Busy := FALSE, Translation_Done := TRUE,
       Benne_Busy := FALSE, Benne_Done := FALSE, Benne_IsOpen := FALSE, Benne_IsClosed := TRUE, Benne_IsRoughlyClosed := TRUE,
       SampleCount := SampleCount);
    (* X3 -> X4 *)
    FB(Enable := TRUE, Reset := FALSE, PowerContactorEngaged := TRUE, Mode := E_Mode.SEMI_AUTO,
       DeadmanArmed := TRUE, CycleMotionPermit := TRUE, HeartbeatIhmOk := TRUE,
       StartCycle := FALSE, SelTarget := 3, SetDepthM := -10.0, SetOffsetM := 0.0,
       LimitLegalDepthM := -10.5, CableLimitM1AscentM := 7.0,
       SpeedMismatchThresholdMps := 0.0, SpeedMismatchTimeout := T#0ms,
       HomedM1 := TRUE, HomedM2 := TRUE, TopPositionSensor := TRUE, HomingRequest := FALSE,
       M1_CablePosM := 7.0, M2_CablePosM := 7.0, M1_MeasuredSpeedMps := 0.0, M2_MeasuredSpeedMps := 0.0,
       KoboldContactFond := FALSE, WinchSyncError := FALSE, WinchSyncDeltaM := 0.0,
       Translation_At_P1 := TRUE, Translation_At_Tremie := FALSE, Translation_At_Maintenance := FALSE,
       Translation_Busy := FALSE, Translation_Done := TRUE,
       Benne_Busy := FALSE, Benne_Done := FALSE, Benne_IsOpen := TRUE, Benne_IsClosed := FALSE, Benne_IsRoughlyClosed := FALSE,
       SampleCount := SampleCount);
    (* X4 (stabilisation) *)
    FB(Enable := TRUE, Reset := FALSE, PowerContactorEngaged := TRUE, Mode := E_Mode.SEMI_AUTO,
       DeadmanArmed := TRUE, CycleMotionPermit := TRUE, HeartbeatIhmOk := TRUE,
       StartCycle := FALSE, SelTarget := 3, SetDepthM := -10.0, SetOffsetM := 0.0,
       LimitLegalDepthM := -10.5, CableLimitM1AscentM := 7.0,
       SpeedMismatchThresholdMps := 0.0, SpeedMismatchTimeout := T#0ms,
       HomedM1 := TRUE, HomedM2 := TRUE, TopPositionSensor := TRUE, HomingRequest := FALSE,
       M1_CablePosM := 7.0, M2_CablePosM := 7.0, M1_MeasuredSpeedMps := 0.0, M2_MeasuredSpeedMps := 0.0,
       KoboldContactFond := FALSE, WinchSyncError := FALSE, WinchSyncDeltaM := 0.0,
       Translation_At_P1 := TRUE, Translation_At_Tremie := FALSE, Translation_At_Maintenance := FALSE,
       Translation_Busy := FALSE, Translation_Done := TRUE,
       Benne_Busy := FALSE, Benne_Done := FALSE, Benne_IsOpen := TRUE, Benne_IsClosed := FALSE, Benne_IsRoughlyClosed := FALSE,
       SampleCount := SampleCount);
    (* Bascule MAINT *)
    FB(Enable := FALSE, Reset := FALSE, PowerContactorEngaged := TRUE, Mode := E_Mode.MAINT_N1,
       DeadmanArmed := TRUE, CycleMotionPermit := TRUE, HeartbeatIhmOk := TRUE,
       StartCycle := FALSE, SelTarget := 3, SetDepthM := -10.0, SetOffsetM := 0.0,
       LimitLegalDepthM := -10.5, CableLimitM1AscentM := 7.0,
       SpeedMismatchThresholdMps := 0.0, SpeedMismatchTimeout := T#0ms,
       HomedM1 := TRUE, HomedM2 := TRUE, TopPositionSensor := TRUE, HomingRequest := FALSE,
       M1_CablePosM := 7.0, M2_CablePosM := 7.0, M1_MeasuredSpeedMps := 0.0, M2_MeasuredSpeedMps := 0.0,
       KoboldContactFond := FALSE, WinchSyncError := FALSE, WinchSyncDeltaM := 0.0,
       Translation_At_P1 := TRUE, Translation_At_Tremie := FALSE, Translation_At_Maintenance := FALSE,
       Translation_Busy := FALSE, Translation_Done := TRUE,
       Benne_Busy := FALSE, Benne_Done := FALSE, Benne_IsOpen := TRUE, Benne_IsClosed := FALSE, Benne_IsRoughlyClosed := FALSE,
       SampleCount := SampleCount);
    (* Retour SEMI_AUTO avec manche défléchi : PAS de mouvement spontané (sur original : mouvement auto) *)
    FB(Enable := TRUE, Reset := FALSE, PowerContactorEngaged := TRUE, Mode := E_Mode.SEMI_AUTO,
       DeadmanArmed := TRUE, CycleMotionPermit := TRUE, HeartbeatIhmOk := TRUE,
       StartCycle := FALSE, SelTarget := 3, SetDepthM := -10.0, SetOffsetM := 0.0,
       LimitLegalDepthM := -10.5, CableLimitM1AscentM := 7.0,
       SpeedMismatchThresholdMps := 0.0, SpeedMismatchTimeout := T#0ms,
       HomedM1 := TRUE, HomedM2 := TRUE, TopPositionSensor := TRUE, HomingRequest := FALSE,
       M1_CablePosM := 7.0, M2_CablePosM := 7.0, M1_MeasuredSpeedMps := 0.0, M2_MeasuredSpeedMps := 0.0,
       KoboldContactFond := FALSE, WinchSyncError := FALSE, WinchSyncDeltaM := 0.0,
       Translation_At_P1 := TRUE, Translation_At_Tremie := FALSE, Translation_At_Maintenance := FALSE,
       Translation_Busy := FALSE, Translation_Done := TRUE,
       Benne_Busy := FALSE, Benne_Done := FALSE, Benne_IsOpen := TRUE, Benne_IsClosed := FALSE, Benne_IsRoughlyClosed := FALSE,
       SampleCount := SampleCount);
    ASSERT_FALSE(FB.WinchM1Cmd.StartStop, 'NEG-F6: PAS de mouvement spontané au retour (échoue sur original)');
END_TEST
